{attribute 'GeneratedUsingTerminal: EP9521-0020-0000'}
{attribute addProperty BoxType "EP9521-0020-0000"}
{attribute addProperty Id "EtcSlaveTerminalBaseInfoDataAT %I*InfoData_6F19DB2B2"}
{attribute addProperty CRC "2874840167"}
{attribute addProperty Size "2"}
TYPE EP9521_AB5A9467 EXTENDS EtcSlaveTerminalBase :
STRUCT
	{attribute addProperty Name "InfoData"}
	InfoData : InfoData_6F19DB2B;
END_STRUCT
END_TYPE

(* stored: Version 1.2.0.0, ProductVersion 3.1.4024.9
   DUT EP9521_AB5A9467: Id {be86cee6-a126-497a-a851-73ab42d9f750} *)
